(* PLC project Logging example, Unknown Generic PLC 1 *)
(* stored: creationDateTime 2013-01-29T14:01:00, contentDescription This example shows logging functionality in Beremiz. Here are shown two ways of logging: - from IEC PLC program; - from python extension., modificationDateTime 2018-08-24T13:12:45 *)

PROGRAM program0
  VAR
    beat : BOOL;
    count : INT;
    LOGGER0 : LOGGER;
    lvl : LOGLEVEL := INFO;
    Timer : TOF;
  END_VAR
  VAR  (* added by the conversion: wires and edge detectors of the diagram *)
    _NOT3_OUT : BOOL;
    R_TRIG1 : R_TRIG;
    _ADD5_OUT : INT;
  END_VAR

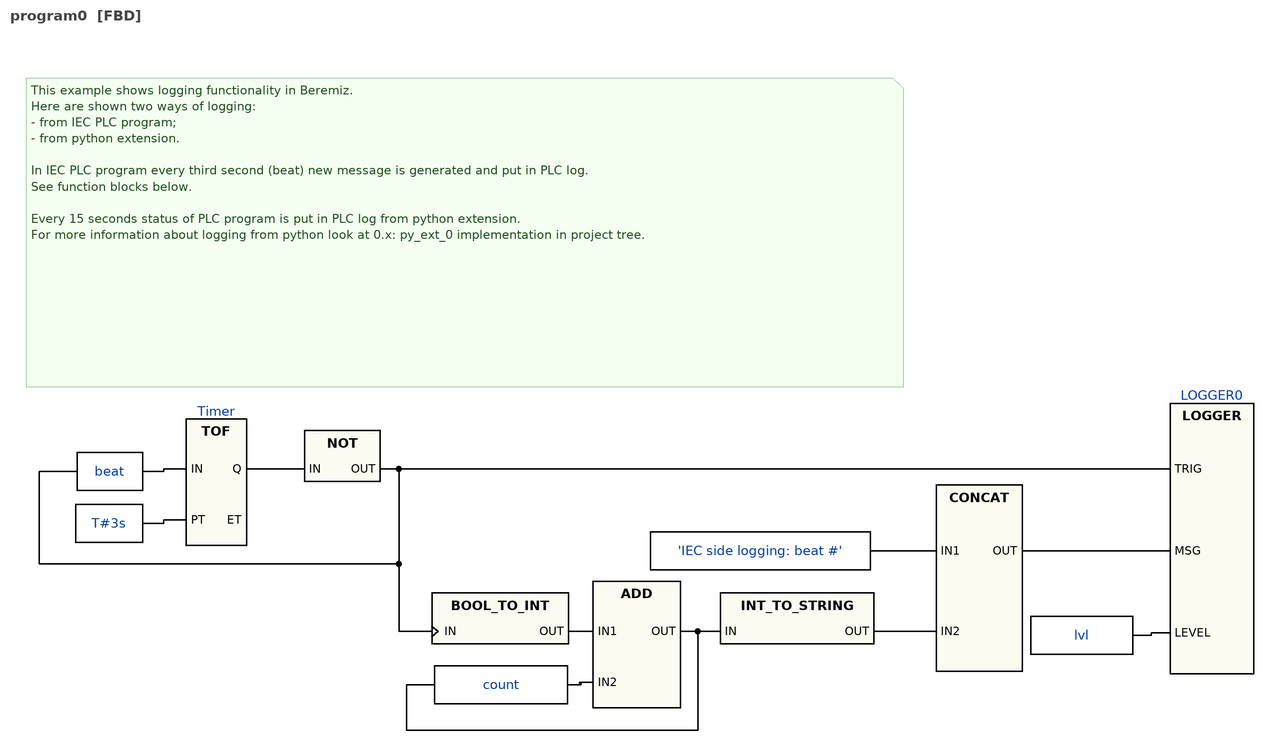
(* FBD diagram, written out as Structured Text *)
(* This example shows logging functionality in Beremiz.
Here are shown two ways of logging:
- from IEC PLC program;
- from python extension.

In IEC PLC program every third second (beat) new message is generated and put in PLC log.
See function blocks below.

Every 15 seconds status of PLC program is put in PLC log from python extension.
For more information about logging from python look at 0.x: py_ext_0 implementation in project tree. *)
Timer(IN := beat, PT := T#3s);
_NOT3_OUT := NOT Timer.Q;
beat := _NOT3_OUT;
R_TRIG1(CLK := _NOT3_OUT);
_ADD5_OUT := BOOL_TO_INT(R_TRIG1.Q) + count;
count := _ADD5_OUT;
LOGGER0(TRIG := _NOT3_OUT, MSG := CONCAT('IEC side logging: beat #', INT_TO_STRING(_ADD5_OUT)), LEVEL := lvl);
END_PROGRAM

CONFIGURATION config
  RESOURCE resource1 ON PLC
    TASK task0(INTERVAL := T#100ms, PRIORITY := 0);
    PROGRAM prg WITH task0 : program0;
  END_RESOURCE
END_CONFIGURATION
